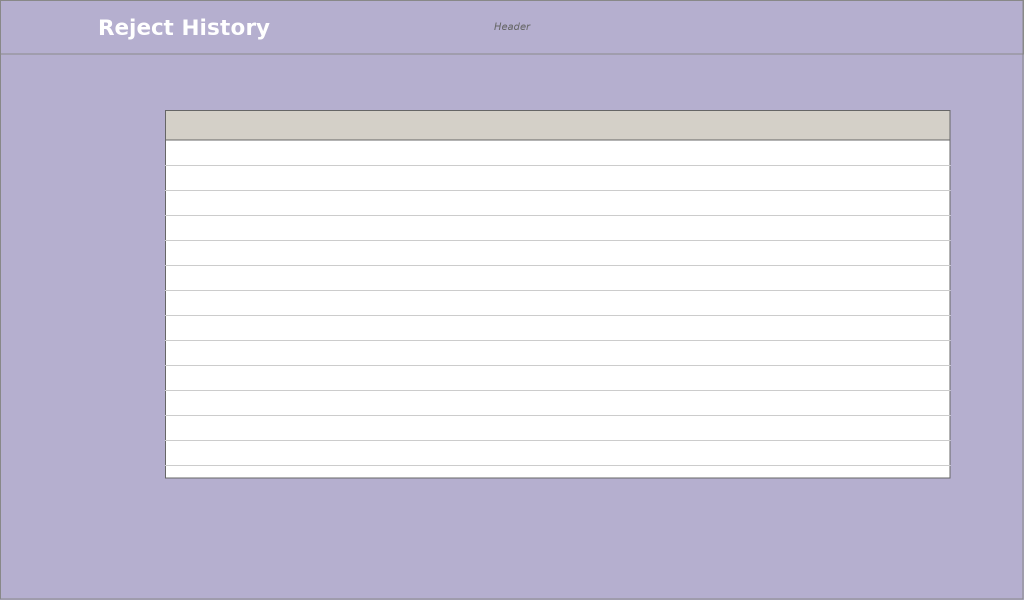
VISUALIZATION RejectMsg  // 1024x600
    Frame (0,-1 1024x55)
        shows Header()
    Label (95,15 250x25), "Reject History"
    Table (165,110 785x368), data array: Status_GVL.arRejectMsg
        p3854506369: Status_GVL.arRejectMsg[INDEX].Status
        p1892666644: Status_GVL.arRejectMsg[INDEX].RejectID
        p338671338: Status_GVL.arRejectMsg[INDEX].RejectType
        p2170511999: Status_GVL.arRejectMsg[INDEX].Counter
        p511219082: Reject ID
        p3723444502: Status_GVL.arRejectMsg[INDEX].RejectMsg
        p1218418051: Status_GVL.arRejectMsg[INDEX].Timestamp
        p2237128397: Message
END_VISUALIZATION

(* stored: Version 1.1.0.1, ProductVersion 3.1.4024.12
   Visu RejectMsg: Id {f76cde95-2904-4f7b-84b4-0534dafc384e} *)
